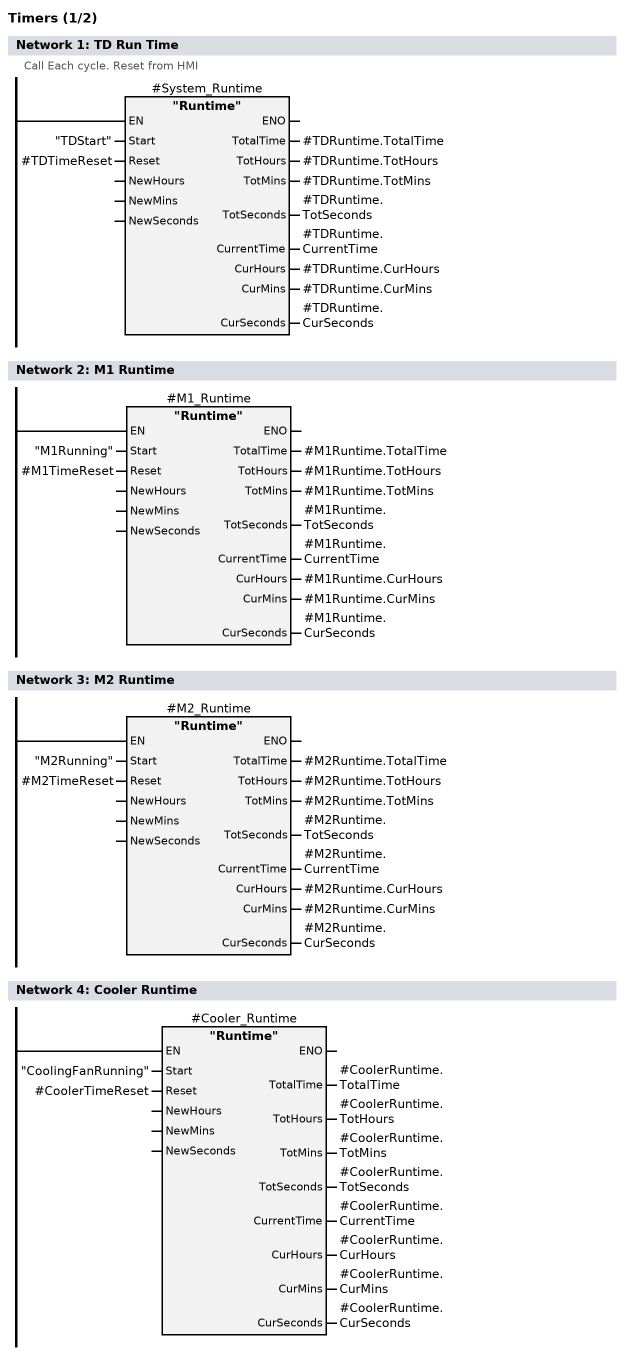
   RUNG wire#powerrail
      #System_Runtime(Start := "TDStart", Reset := #TDTimeReset, NewHours :=, NewMins :=, NewSeconds :=, TotalTime => #TDRuntime.TotalTime, TotHours => #TDRuntime.TotHours, TotMins => #TDRuntime.TotMins, TotSeconds => #TDRuntime.TotSeconds, CurrentTime => #TDRuntime.CurrentTime, CurHours => #TDRuntime.CurHours, CurMins => #TDRuntime.CurMins, CurSeconds => #TDRuntime.CurSeconds)
   END_RUNG
   // the same network as SCL:
   #System_Runtime(Start := "TDStart",   // "Runtime"
                   Reset := #TDTimeReset,
                   TotalTime => #TDRuntime.TotalTime,
                   TotHours => #TDRuntime.TotHours,
                   TotMins => #TDRuntime.TotMins,
                   TotSeconds => #TDRuntime.TotSeconds,
                   CurrentTime => #TDRuntime.CurrentTime,
                   CurHours => #TDRuntime.CurHours,
                   CurMins => #TDRuntime.CurMins,
                   CurSeconds => #TDRuntime.CurSeconds);
END_REGION

REGION Network 2: M1 Runtime
   RUNG wire#powerrail
      #M1_Runtime(Start := "M1Running", Reset := #M1TimeReset, NewHours :=, NewMins :=, NewSeconds :=, TotalTime => #M1Runtime.TotalTime, TotHours => #M1Runtime.TotHours, TotMins => #M1Runtime.TotMins, TotSeconds => #M1Runtime.TotSeconds, CurrentTime => #M1Runtime.CurrentTime, CurHours => #M1Runtime.CurHours, CurMins => #M1Runtime.CurMins, CurSeconds => #M1Runtime.CurSeconds)
   END_RUNG
   // the same network as SCL:
   #M1_Runtime(Start := "M1Running",   // "Runtime"
               Reset := #M1TimeReset,
               TotalTime => #M1Runtime.TotalTime,
               TotHours => #M1Runtime.TotHours,
               TotMins => #M1Runtime.TotMins,
               TotSeconds => #M1Runtime.TotSeconds,
               CurrentTime => #M1Runtime.CurrentTime,
               CurHours => #M1Runtime.CurHours,
               CurMins => #M1Runtime.CurMins,
               CurSeconds => #M1Runtime.CurSeconds);
END_REGION

REGION Network 3: M2 Runtime
   RUNG wire#powerrail
      #M2_Runtime(Start := "M2Running", Reset := #M2TimeReset, NewHours :=, NewMins :=, NewSeconds :=, TotalTime => #M2Runtime.TotalTime, TotHours => #M2Runtime.TotHours, TotMins => #M2Runtime.TotMins, TotSeconds => #M2Runtime.TotSeconds, CurrentTime => #M2Runtime.CurrentTime, CurHours => #M2Runtime.CurHours, CurMins => #M2Runtime.CurMins, CurSeconds => #M2Runtime.CurSeconds)
   END_RUNG
   // the same network as SCL:
   #M2_Runtime(Start := "M2Running",   // "Runtime"
               Reset := #M2TimeReset,
               TotalTime => #M2Runtime.TotalTime,
               TotHours => #M2Runtime.TotHours,
               TotMins => #M2Runtime.TotMins,
               TotSeconds => #M2Runtime.TotSeconds,
               CurrentTime => #M2Runtime.CurrentTime,
               CurHours => #M2Runtime.CurHours,
               CurMins => #M2Runtime.CurMins,
               CurSeconds => #M2Runtime.CurSeconds);
END_REGION

REGION Network 4: Cooler Runtime
   RUNG wire#powerrail
      #Cooler_Runtime(Start := "CoolingFanRunning", Reset := #CoolerTimeReset, NewHours :=, NewMins :=, NewSeconds :=, TotalTime => #CoolerRuntime.TotalTime, TotHours => #CoolerRuntime.TotHours, TotMins => #CoolerRuntime.TotMins, TotSeconds => #CoolerRuntime.TotSeconds, CurrentTime => #CoolerRuntime.CurrentTime, CurHours => #CoolerRuntime.CurHours, CurMins => #CoolerRuntime.CurMins, CurSeconds => #CoolerRuntime.CurSeconds)
   END_RUNG
   // the same network as SCL:
   #Cooler_Runtime(Start := "CoolingFanRunning",   // "Runtime"
                   Reset := #CoolerTimeReset,
                   TotalTime => #CoolerRuntime.TotalTime,
                   TotHours => #CoolerRuntime.TotHours,
                   TotMins => #CoolerRuntime.TotMins,
                   TotSeconds => #CoolerRuntime.TotSeconds,
                   CurrentTime => #CoolerRuntime.CurrentTime,
                   CurHours => #CoolerRuntime.CurHours,
                   CurMins => #CoolerRuntime.CurMins,
                   CurSeconds => #CoolerRuntime.CurSeconds);
END_REGION

REGION Network 5: Aux Pump Runtime
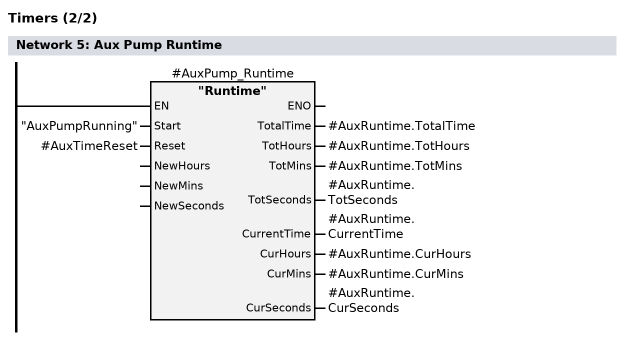
   RUNG wire#powerrail
      #AuxPump_Runtime(Start := "AuxPumpRunning", Reset := #AuxTimeReset, NewHours :=, NewMins :=, NewSeconds :=, TotalTime => #AuxRuntime.TotalTime, TotHours => #AuxRuntime.TotHours, TotMins => #AuxRuntime.TotMins, TotSeconds => #AuxRuntime.TotSeconds, CurrentTime => #AuxRuntime.CurrentTime, CurHours => #AuxRuntime.CurHours, CurMins => #AuxRuntime.CurMins, CurSeconds => #AuxRuntime.CurSeconds)
   END_RUNG
   // the same network as SCL:
   #AuxPump_Runtime(Start := "AuxPumpRunning",   // "Runtime"
                    Reset := #AuxTimeReset,
                    TotalTime => #AuxRuntime.TotalTime,
                    TotHours => #AuxRuntime.TotHours,
                    TotMins => #AuxRuntime.TotMins,
                    TotSeconds => #AuxRuntime.TotSeconds,
                    CurrentTime => #AuxRuntime.CurrentTime,
                    CurHours => #AuxRuntime.CurHours,
                    CurMins => #AuxRuntime.CurMins,
                    CurSeconds => #AuxRuntime.CurSeconds);
END_REGION
END_FUNCTION_BLOCK

FUNCTION_BLOCK "Runtime"   // FB124, LAD
{ S7_Optimized_Access := 'TRUE' }
// Written By Kristopher Gimenez March 3rd,2023
// 
// This block and its DB will perform a runtime counter and outputs total runtime in Hours, Minutes and Seconds
// stored: AutoNumber false, MemoryReserve 100, SetENOAutomatically false
   VAR_INPUT
      Start : Bool;
      Reset : Bool;
      NewHours : DInt;
      NewMins : DInt;
      NewSeconds : DInt;
   END_VAR
   VAR_OUTPUT
      TotalTime : DInt;
      TotHours : DInt;
      TotMins : DInt;
      TotSeconds : DInt;
      CurrentTime : DInt;   // Current Time in Seconds
      CurHours : DInt;
      CurMins : DInt;
      CurSeconds : DInt;
   END_VAR
   VAR
      StartTrig : Bool;
      StartTime : DInt;
      Runtime_TONR { S7_SetPoint := 'True'} : TONR_TIME;
      TimerReset { ExternalAccessible := 'False'; ExternalVisible := 'False'; ExternalWritable := 'False'} : Bool;
      CurrentIECTime : Time;
      NewTime : DInt;   // New Time in seconds to reset to base on inputs
   END_VAR
   VAR_TEMP
      TempDInt : DInt;
      NewHoursInSec : DInt;
      NewMinsInSec : DInt;
   END_VAR
   VAR_TEMP   // added for the SCL form of the ladder/FBD networks
      _w1 : Bool;
   END_VAR
BEGIN

REGION Network 1: Start
   // When Starting store Total as Start Value
   // Reset Current Runtime
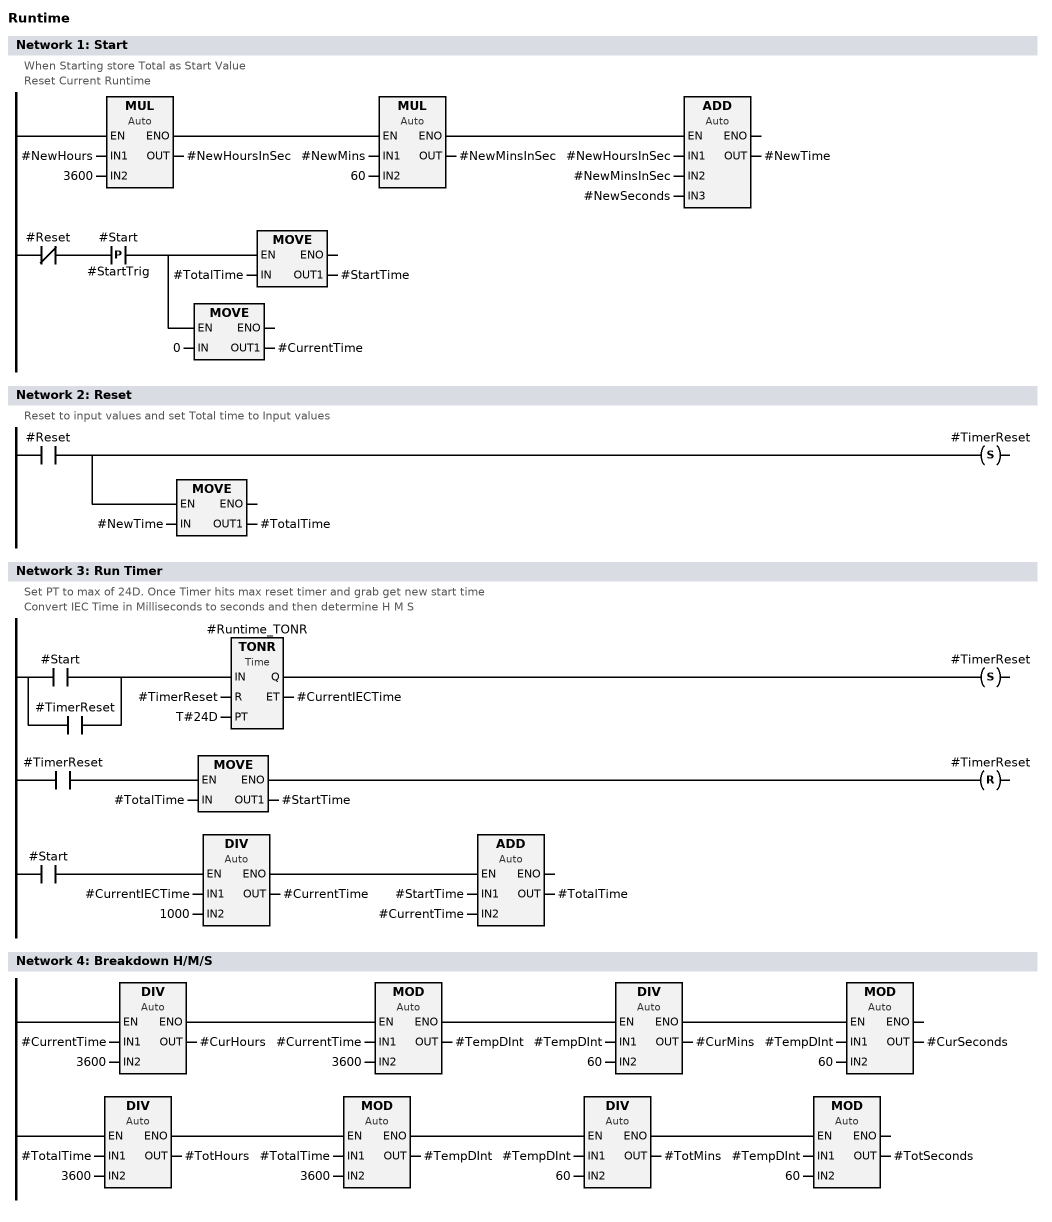
   RUNG wire#powerrail
      Mul(in1 := #NewHours, in2 := 3600, out => #NewHoursInSec)
      Mul(in1 := #NewMins, in2 := 60, out => #NewMinsInSec)
      Add(in1 := #NewHoursInSec, in2 := #NewMinsInSec, in3 := #NewSeconds, out => #NewTime)
   END_RUNG
   RUNG wire#powerrail
      I_Contact( #Reset )
      P_Contact(operand := #Start, bit := #StartTrig)
      wire#w1
      Move(in := #TotalTime, out1 => #StartTime)
   END_RUNG
   RUNG wire#w1
      Move(in := 0, out1 => #CurrentTime)
   END_RUNG
   // the same network as SCL:
   #NewHoursInSec := #NewHours * 3600;
   #NewMinsInSec := #NewMins * 60;
   #NewTime := #NewHoursInSec + #NewMinsInSec + #NewSeconds;
   #_w1 := NOT #Reset AND #Start AND NOT #StartTrig;   // rising edge of #Start
   #StartTrig := #Start;
   IF #_w1 THEN
       #StartTime := #TotalTime;
       #CurrentTime := 0;
   END_IF;
END_REGION

REGION Network 2: Reset
   // Reset to input values and set Total time to Input values
   RUNG wire#powerrail
      Contact( #Reset )
      wire#w1
      S_Coil( #TimerReset )
   END_RUNG
   RUNG wire#w1
      Move(in := #NewTime, out1 => #TotalTime)
   END_RUNG
   // the same network as SCL:
   IF #Reset THEN
       #TimerReset := TRUE;
       #TotalTime := #NewTime;
   END_IF;
END_REGION

REGION Network 3: Run Timer
   // Set PT to max of 24D. Once Timer hits max reset timer and grab get new start time
   // Convert IEC Time in Milliseconds to seconds and then determine H M S
   RUNG wire#powerrail
      Contact( #Start )
      wire#w1
      { S7_Templates := "time_type := Time" } #Runtime_TONR.TONR(r := #TimerReset, pt := T#24D, et => #CurrentIECTime)
      S_Coil( #TimerReset )
   END_RUNG
   RUNG wire#powerrail
      Contact( #TimerReset )
   END_RUNG wire#w1
   RUNG wire#powerrail
      Contact( #TimerReset )
      Move(in := #TotalTime, out1 => #StartTime)
      R_Coil( #TimerReset )
   END_RUNG
   RUNG wire#powerrail
      Contact( #Start )
      Div(in1 := #CurrentIECTime, in2 := 1000, out => #CurrentTime)
      Add(in1 := #StartTime, in2 := #CurrentTime, out => #TotalTime)
   END_RUNG
   // the same network as SCL:
   #Runtime_TONR(IN := #Start OR #TimerReset, R := #TimerReset, PT := T#24D, ET => #CurrentIECTime);   // TONR
   IF #Runtime_TONR.Q THEN #TimerReset := TRUE; END_IF;
   IF #TimerReset THEN
       #StartTime := #TotalTime;
       #TimerReset := FALSE;
   END_IF;
   IF #Start THEN
       #CurrentTime := #CurrentIECTime / 1000;
       #TotalTime := #StartTime + #CurrentTime;
   END_IF;
END_REGION

REGION Network 4: Breakdown H/M/S
   RUNG wire#powerrail
      Div(in1 := #CurrentTime, in2 := 3600, out => #CurHours)
      Mod(in1 := #CurrentTime, in2 := 3600, out => #TempDInt)
      Div(in1 := #TempDInt, in2 := 60, out => #CurMins)
      Mod(in1 := #TempDInt, in2 := 60, out => #CurSeconds)
   END_RUNG
   RUNG wire#powerrail
      Div(in1 := #TotalTime, in2 := 3600, out => #TotHours)
      Mod(in1 := #TotalTime, in2 := 3600, out => #TempDInt)
      Div(in1 := #TempDInt, in2 := 60, out => #TotMins)
      Mod(in1 := #TempDInt, in2 := 60, out => #TotSeconds)
   END_RUNG
   // the same network as SCL:
   #CurHours := #CurrentTime / 3600;
   #TempDInt := #CurrentTime MOD 3600;
   #CurMins := #TempDInt / 60;
   #CurSeconds := #TempDInt MOD 60;
   #TotHours := #TotalTime / 3600;
   #TempDInt := #TotalTime MOD 3600;
   #TotMins := #TempDInt / 60;
   #TotSeconds := #TempDInt MOD 60;
END_REGION
END_FUNCTION_BLOCK

FUNCTION "MapConsoleOutputs" : Void
{ S7_Optimized_Access := 'TRUE' }
VERSION : 0.1

BEGIN
	(* #MapConsoleOutputs Written BY Kristopher Gimenez January 23,2023
	This block is will map the output variables and convert raw signals into measured values
	*)
	
	
	
	//Slot 4 16x Digital Outputs
	"Console_Out".Slot4.Ch0 :="PTOLED";
	"Console_Out".Slot4.Ch1 := "HPUFaultLED";
	"Console_Out".Slot4.Ch2 := "TDFlushFaultLED";
	"Console_Out".Slot4.Ch3 := "BUWClLED";
	"Console_Out".Slot4.Ch4 := "TDEnLED";
	"Console_Out".Slot4.Ch5 := "ConLowPurgeLED";
	"Console_Out".Slot4.Ch6 := "MSVClLED";
	"Console_Out".Slot4.Ch7 := "QuillLockLED";
	"Console_Out".Slot4.Ch8 := "ElevClLED";
	"Console_Out".Slot4.Ch9 := "Horn";
	"Console_Out".Slot4.Ch10 := "MSVClInt";
	"Console_Out".Slot4.Ch11 := "BUWClInt";
	(*Spare Outputs
	"Console_Out".Slot4.Ch12 := ;
	"Console_Out".Slot4.Ch13 := ;
	"Console_Out".Slot4.Ch14 := ;
	"Console_Out".Slot4.Ch15 := ;
	*)
	
	
	
	
	//Slot 5 4 x AQ U/I
	"AoUI_Scaling"(Measured:="DrillRecTorqFtLbs",
	               Max:=40000.0,
	               Min:=0,
	               s7Raw=>"DrillRecTorqRaw",
	               mAOutput=>"DrillRecTorqmA"); //4-20ma = 0-40 000 ft-lbs
	"AoUI_Scaling"(Measured:="DrillRecRPM",
	               Max:=200.0,
	               Min:=0,
	               s7Raw=>"DrillRecRPMRaw",
	               mAOutput=>"DrillRecRPMmA");// 4-20ma = 0-200 RPM
	
	
	"Console_Out".Slot5.Ch0 := "DrillRecTorqRaw";
	"Console_Out".Slot5.Ch1 := ("DrillRecRPMRaw");
END_FUNCTION

FUNCTION "AoUI_Scaling" : Void
{ S7_Optimized_Access := 'TRUE' }
VERSION : 0.1
   VAR_INPUT 
      Measured : Real;   // Measured
      Max : Real;   // Maximum mreasured value of output
      Min : Real;   // Minimum measured value of output
   END_VAR

   VAR_OUTPUT 
      s7Raw : Int;   // Raw Outputs to card 
      mAOutput : Real;   // 4-20ma Output based on raw outputs
   END_VAR


BEGIN
	(* #AoUI_Scaling Written BY Kristopher Gimenez January 23,2023
	This block is used to convert a Measured value into a PS7 analog output and the corresponding 4-20mA signal based on Scale and Offset. 
	*)
	
	
	#s7Raw := REAL_TO_INT((#Measured-#Min)/(#Max - #Min) * 27648);
	#mAOutput := ((#Measured-#Min)/(#Max-#Min) * 16.0) + 4.0;
	
	
END_FUNCTION

FUNCTION "MapHPUOutputs" : Void
{ S7_Optimized_Access := 'TRUE' }
VERSION : 0.1

BEGIN
	(* #MapHPUOutputs Written BY Kristopher Gimenez January 19,2023
	This block is will map the input variables and convert raw signals into measured values
	*)
	//HPU Slot2 TM Count Encoder Outputs
	"HPU_Out".Slot2.SW_GATE := "SwitchSWGATE"; //Enable the counter
	"HPU_Out".Slot2.SET_DIR:= "RotaryEncInvDir";
	"HPU_Out".Slot2.SLOT_0 := "RotEncSlot0";
	"HPU_Out".Slot2.SLOT_1 := "RotEncSlot1";
	"HPU_Out".Slot2.LD_SLOT_0_1 := "RotEncLDSlot";//assign loading bytes
	"HPU_Out".Slot2.RES_EVENT := "RotEncPosReset";//reset event flags if position is being res
	
	
	//Slot 7 TM Pulse
	//Channel 0 TD P1 Fwd
	"TDFwdPress1Raw" := "AoP_mA2Raw_2A"("TDFwdPress1mA");
	"HPU_Out".Slot7.Ch0.OUTPUT_VALUE := "TDFwdPress1Raw";//assign output value
	"HPU_Out".Slot7.Ch0.SW_ENABLE :="TDFwdPress1En"; //used to enabled output
	"HPU_Out".Slot7.Ch0.DITHER := "TDFwdPress1En"; //enable Dither - Currently enabling with the output. 
	"HPU_Out".Slot7.Ch0.TM_CTRL_DQ :=1;//enable technology control of outputs 
	//Channel 1 TD P1 Rev
	"TDRevPress1Raw" := "AoP_mA2Raw_2A"("TDRevPress1mA");
	"HPU_Out".Slot7.Ch1.OUTPUT_VALUE := "TDRevPress1Raw";//assign output value
	"HPU_Out".Slot7.Ch1.SW_ENABLE := "TDRevPress1En"; //used to enabled output
	"HPU_Out".Slot7.Ch1.DITHER := "TDRevPress1En"; //enable Dither - Currently enabling with the output. 
	"HPU_Out".Slot7.Ch1.TM_CTRL_DQ := 1;//enable technology control of outputs 
	
	
	
	//Slot 8 TM Pulse
	//Channel 0 TD P2 FWD
	"TDFwdPress2Raw" := "AoP_mA2Raw_2A"("TDFwdPress2mA");
	"HPU_Out".Slot8.Ch0.OUTPUT_VALUE := "TDFwdPress2Raw";//assign output value
	"HPU_Out".Slot8.Ch0.SW_ENABLE := "TDFwdPress2En"; //used to enabled output
	"HPU_Out".Slot8.Ch0.DITHER := "TDFwdPress2En"; //enable Dither - Currently enabling with the output. 
	"HPU_Out".Slot8.Ch0.TM_CTRL_DQ := 1;//enable technology control of outputs 
	
	//Channel 1 TD P2 Rev
	"TDRevPress2Raw" := "AoP_mA2Raw_2A"("TDRevPress2mA");
	"HPU_Out".Slot8.Ch1.OUTPUT_VALUE := "TDRevPress2Raw";//assign output value
	"HPU_Out".Slot8.Ch1.SW_ENABLE := "TDRevPress2En"; //used to enabled output
	"HPU_Out".Slot8.Ch1.DITHER := "TDRevPress2En"; //enable Dither - Currently enabling with the output. 
	"HPU_Out".Slot8.Ch1.TM_CTRL_DQ := 1;//enable technology control of outputs 
	
	
	//Slot 9 TM Pulse
	//Channel 0 TD Torq
	"TDTorqPressRaw" := "AoP_mA2Raw_2A"("TDTorqPressmA");
	"HPU_Out".Slot9.Ch0.OUTPUT_VALUE := "TDTorqPressRaw";//assign output value
	"HPU_Out".Slot9.Ch0.SW_ENABLE := "TDTorqPressEn"; //used to enabled output
	"HPU_Out".Slot9.Ch0.DITHER := "TDTorqPressEn"; //enable Dither - Currently enabling with the output. 
	"HPU_Out".Slot9.Ch0.TM_CTRL_DQ := 1;//enable technology control of outputs 
	//Slot 9 TM Pulse
	//Channel 1 TD P1 Rev
	//"TDRevPress1Raw" := "AoP_mA2Raw_2A"("TDRevPress1mA");
	//"HPU_Out".Slot9.Ch1.OUTPUT_VALUE := "TDRevPress1Raw";//assign output value
	//"HPU_Out".Slot9.Ch1.SW_ENABLE := "TDRevPress1En"; //used to enabled output
	//"HPU_Out".Slot9.Ch1.DITHER := "TDRevPress1En"; //enable Dither - Currently enabling with the output. 
	//"HPU_Out".Slot9.Ch1.TM_CTRL_DQ := 1;//enable technology control of outputs 
	
	//Slot 10 DO Relay x 4
	"HPU_Out".Slot10.Ch0 := "M1Start";
	"HPU_Out".Slot10.Ch1 := "M2Start";
	"HPU_Out".Slot10.Ch2 := "CoolingFanStart";
	"HPU_Out".Slot10.Ch3 := "AuxPumpStart";
	
	//Slot 11 DO Relay x 4
	"HPU_Out".Slot11.Ch0 := "LinkExtSol";
	"HPU_Out".Slot11.Ch1 := "LinkRetSol";
	"HPU_Out".Slot11.Ch2 := "LinkFloatSol";
	//"HPU_Out".Slot11.Ch3 := ;Spare
	
	
	//Slot 12 DO Relay x 4
	"HPU_Out".Slot12.Ch0 := "BUWClSol";
	"HPU_Out".Slot12.Ch1 := "BUWDnSol";
	"HPU_Out".Slot12.Ch2 := "BUWUpSol";
	"HPU_Out".Slot12.Ch3 := "BUWOpSol";
	
	
	//Slot 13 DO Relay x 4
	"HPU_Out".Slot13.Ch0 := "LSHT_Sol";
	"HPU_Out".Slot13.Ch1 := "HSLT_Sol";
	"HPU_Out".Slot13.Ch2 := "ElevClSol";
	"HPU_Out".Slot13.Ch3 := "ElevOpSol";
	
	
	//Slot 14 DO Relay x 4
	"HPU_Out".Slot14.Ch0 := "HandlerFWDSol";
	"HPU_Out".Slot14.Ch1 := "HandlerREVSol";
	"HPU_Out".Slot14.Ch2 := "MSVOpSol";
	"HPU_Out".Slot14.Ch3 := "MSVClSol";
	
	
	//Slot 15 DO Relay x 4
	"HPU_Out".Slot15.Ch0 := "HourMeterOn";
	"HPU_Out".Slot15.Ch1 := "FailSafeEnSol";
	"HPU_Out".Slot15.Ch2 := "AuxUnloaderSol";
	"HPU_Out".Slot15.Ch3 := "BypassValveSol";
	
	
	//Slot 16 DO Relay x 4
	"HPU_Out".Slot16.Ch0 := "TDExtSol";
	"HPU_Out".Slot16.Ch1 := "TDRetSol";
	"HPU_Out".Slot16.Ch2 := "HotOilControlSol";
	"HPU_Out".Slot16.Ch3 := "BOControlSol";
	
	//Slot 17 DO Relay x 4
	(*Spare Outputs
	"HPU_Out".Slot17.Ch0 := ;
	"HPU_Out".Slot17.Ch1 := ;
	"HPU_Out".Slot18.Ch2 := ;
	"HPU_Out".Slot18.Ch3 := ;
	*)
END_FUNCTION

FUNCTION "AoP_mA2Raw_2A" : UDInt
{ S7_Optimized_Access := 'TRUE' }
VERSION : 0.1
   VAR_INPUT 
      Realnput : Real;
   END_VAR


BEGIN
	(* #AoP_ma2Raw_2A Written BY Kristopher Gimenez January 23,2023
	This block is used to convert a mA signal  output signal to a Raw. Note 0-2A = 27648 pulse output.
	*)
	
	
	#AoP_mA2Raw_2A := REAL_TO_UDINT(#Realnput/2000* 27648.0);
	
	
END_FUNCTION

ORGANIZATION_BLOCK "Startup"   // OB100, LAD, Startup
TITLE = "Complete Restart"
{ S7_Optimized_Access := 'TRUE' }
// stored: SetENOAutomatically false
   VAR_INPUT
      LostRetentive : Bool;   // True if retentive data are lost
      LostRTC : Bool;   // True if date and time are lost
   END_VAR
   VAR_TEMP
      RetVal : Int;
      BusyStatus : Bool;
   END_VAR
   VAR_TEMP   // added for the SCL form of the ladder/FBD networks
      _w1 : Bool;
   END_VAR
BEGIN

REGION Network 1: Verify Settings
   // Check settings on startup
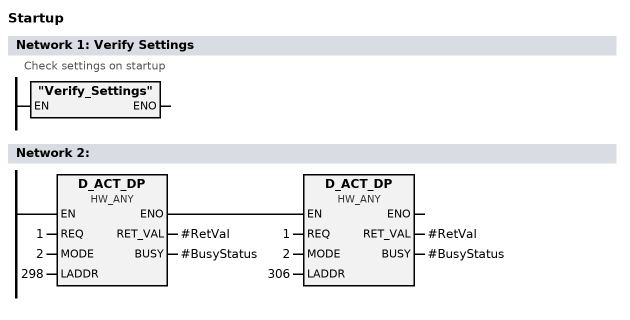
   RUNG wire#powerrail
      "Verify_Settings"()
   END_RUNG
   // the same network as SCL:
   "Verify_Settings"();
END_REGION

REGION Network 2
   RUNG wire#powerrail
      { S7_Templates := "[laddr_type := HW_ANY, mode_type := USInt]" } D_ACT_DP(REQ := 1, MODE := 2, LADDR := 298, RET_VAL => #RetVal, BUSY => #BusyStatus)
      { S7_Templates := "[laddr_type := HW_ANY, mode_type := USInt]" } D_ACT_DP(REQ := 1, MODE := 2, LADDR := 306, RET_VAL => #RetVal, BUSY => #BusyStatus)
   END_RUNG
   // the same network as SCL:
   #RetVal := D_ACT_DP(REQ := 1, MODE := 2, LADDR := 298, BUSY => #BusyStatus, ENO => #_w1);
   IF #_w1 THEN #RetVal := D_ACT_DP(REQ := 1, MODE := 2, LADDR := 306, BUSY => #BusyStatus); END_IF;
END_REGION
END_ORGANIZATION_BLOCK

FUNCTION "Verify_Settings" : Void   // FC21, LAD
{ S7_Optimized_Access := 'TRUE' }
// Written BY Kristopher Gimenez February 9th, 2023
// This block is used to check the settings are within limits and adjust as needed
// stored: AutoNumber false, SetENOAutomatically false
BEGIN

REGION Network 1: Alpha Values
   // All alpha filter values between 0-1
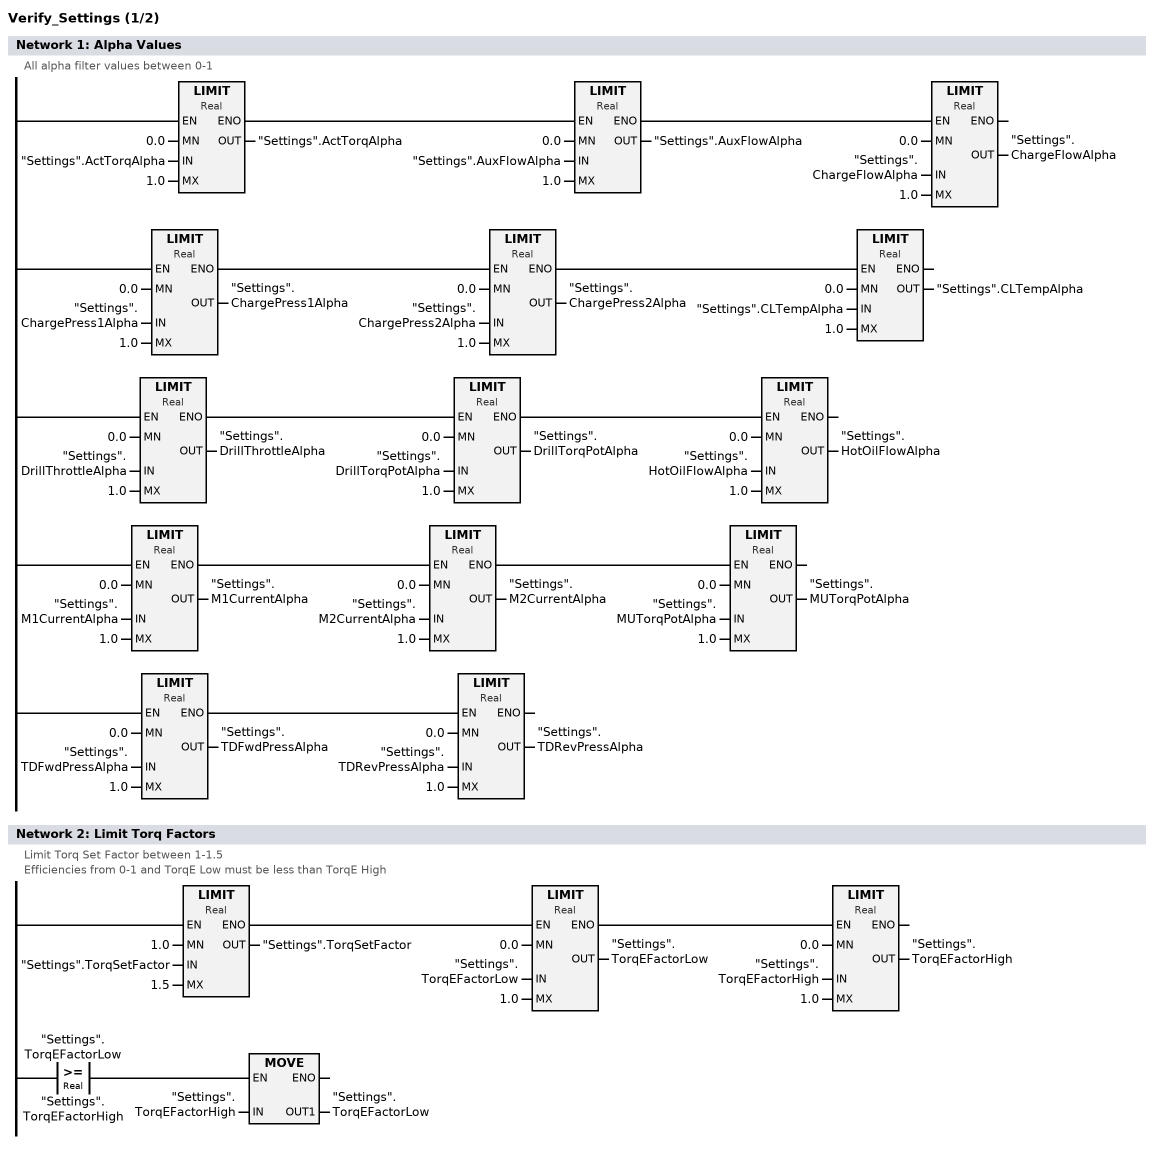
   RUNG wire#powerrail
      { S7_Templates := "value_type := Real" } Limit(mn := 0.0, in := "Settings".ActTorqAlpha, mx := 1.0, out => "Settings".ActTorqAlpha)
      { S7_Templates := "value_type := Real" } Limit(mn := 0.0, in := "Settings".AuxFlowAlpha, mx := 1.0, out => "Settings".AuxFlowAlpha)
      { S7_Templates := "value_type := Real" } Limit(mn := 0.0, in := "Settings".ChargeFlowAlpha, mx := 1.0, out => "Settings".ChargeFlowAlpha)
   END_RUNG
   RUNG wire#powerrail
      { S7_Templates := "value_type := Real" } Limit(mn := 0.0, in := "Settings".ChargePress1Alpha, mx := 1.0, out => "Settings".ChargePress1Alpha)
      { S7_Templates := "value_type := Real" } Limit(mn := 0.0, in := "Settings".ChargePress2Alpha, mx := 1.0, out => "Settings".ChargePress2Alpha)
      { S7_Templates := "value_type := Real" } Limit(mn := 0.0, in := "Settings".CLTempAlpha, mx := 1.0, out => "Settings".CLTempAlpha)
   END_RUNG
   RUNG wire#powerrail
      { S7_Templates := "value_type := Real" } Limit(mn := 0.0, in := "Settings".DrillThrottleAlpha, mx := 1.0, out => "Settings".DrillThrottleAlpha)
      { S7_Templates := "value_type := Real" } Limit(mn := 0.0, in := "Settings".DrillTorqPotAlpha, mx := 1.0, out => "Settings".DrillTorqPotAlpha)
      { S7_Templates := "value_type := Real" } Limit(mn := 0.0, in := "Settings".HotOilFlowAlpha, mx := 1.0, out => "Settings".HotOilFlowAlpha)
   END_RUNG
   RUNG wire#powerrail
      { S7_Templates := "value_type := Real" } Limit(mn := 0.0, in := "Settings".M1CurrentAlpha, mx := 1.0, out => "Settings".M1CurrentAlpha)
      { S7_Templates := "value_type := Real" } Limit(mn := 0.0, in := "Settings".M2CurrentAlpha, mx := 1.0, out => "Settings".M2CurrentAlpha)
      { S7_Templates := "value_type := Real" } Limit(mn := 0.0, in := "Settings".MUTorqPotAlpha, mx := 1.0, out => "Settings".MUTorqPotAlpha)
   END_RUNG
   RUNG wire#powerrail
      { S7_Templates := "value_type := Real" } Limit(mn := 0.0, in := "Settings".TDFwdPressAlpha, mx := 1.0, out => "Settings".TDFwdPressAlpha)
      { S7_Templates := "value_type := Real" } Limit(mn := 0.0, in := "Settings".TDRevPressAlpha, mx := 1.0, out => "Settings".TDRevPressAlpha)
   END_RUNG
   // the same network as SCL:
   "Settings".ActTorqAlpha := LIMIT(MN := 0.0, IN := "Settings".ActTorqAlpha, MX := 1.0);
   "Settings".AuxFlowAlpha := LIMIT(MN := 0.0, IN := "Settings".AuxFlowAlpha, MX := 1.0);
   "Settings".ChargeFlowAlpha := LIMIT(MN := 0.0, IN := "Settings".ChargeFlowAlpha, MX := 1.0);
   "Settings".ChargePress1Alpha := LIMIT(MN := 0.0, IN := "Settings".ChargePress1Alpha, MX := 1.0);
   "Settings".ChargePress2Alpha := LIMIT(MN := 0.0, IN := "Settings".ChargePress2Alpha, MX := 1.0);
   "Settings".CLTempAlpha := LIMIT(MN := 0.0, IN := "Settings".CLTempAlpha, MX := 1.0);
   "Settings".DrillThrottleAlpha := LIMIT(MN := 0.0, IN := "Settings".DrillThrottleAlpha, MX := 1.0);
   "Settings".DrillTorqPotAlpha := LIMIT(MN := 0.0, IN := "Settings".DrillTorqPotAlpha, MX := 1.0);
   "Settings".HotOilFlowAlpha := LIMIT(MN := 0.0, IN := "Settings".HotOilFlowAlpha, MX := 1.0);
   "Settings".M1CurrentAlpha := LIMIT(MN := 0.0, IN := "Settings".M1CurrentAlpha, MX := 1.0);
   "Settings".M2CurrentAlpha := LIMIT(MN := 0.0, IN := "Settings".M2CurrentAlpha, MX := 1.0);
   "Settings".MUTorqPotAlpha := LIMIT(MN := 0.0, IN := "Settings".MUTorqPotAlpha, MX := 1.0);
   "Settings".TDFwdPressAlpha := LIMIT(MN := 0.0, IN := "Settings".TDFwdPressAlpha, MX := 1.0);
   "Settings".TDRevPressAlpha := LIMIT(MN := 0.0, IN := "Settings".TDRevPressAlpha, MX := 1.0);
END_REGION

REGION Network 2: Limit Torq Factors
   // Limit Torq Set Factor between 1-1.5
   // Efficiencies from 0-1 and TorqE Low must be less than TorqE High
   RUNG wire#powerrail
      { S7_Templates := "value_type := Real" } Limit(mn := 1.0, in := "Settings".TorqSetFactor, mx := 1.5, out => "Settings".TorqSetFactor)
      { S7_Templates := "value_type := Real" } Limit(mn := 0.0, in := "Settings".TorqEFactorLow, mx := 1.0, out => "Settings".TorqEFactorLow)
      { S7_Templates := "value_type := Real" } Limit(mn := 0.0, in := "Settings".TorqEFactorHigh, mx := 1.0, out => "Settings".TorqEFactorHigh)
   END_RUNG
   RUNG wire#powerrail
      { S7_Templates := "SrcType := Real" } GE_Contact(in1 := "Settings".TorqEFactorLow, in2 := "Settings".TorqEFactorHigh)
      Move(in := "Settings".TorqEFactorHigh, out1 => "Settings".TorqEFactorLow)
   END_RUNG
   // the same network as SCL:
   "Settings".TorqSetFactor := LIMIT(MN := 1.0, IN := "Settings".TorqSetFactor, MX := 1.5);
   "Settings".TorqEFactorLow := LIMIT(MN := 0.0, IN := "Settings".TorqEFactorLow, MX := 1.0);
   "Settings".TorqEFactorHigh := LIMIT(MN := 0.0, IN := "Settings".TorqEFactorHigh, MX := 1.0);
   IF "Settings".TorqEFactorLow >= "Settings".TorqEFactorHigh THEN
       "Settings".TorqEFactorLow := "Settings".TorqEFactorHigh;
   END_IF;
END_REGION

REGION Network 3: Verify BO Setting
   // BO Spin Factor from 1-2
   // Shift RPM from 1 to Speed limit
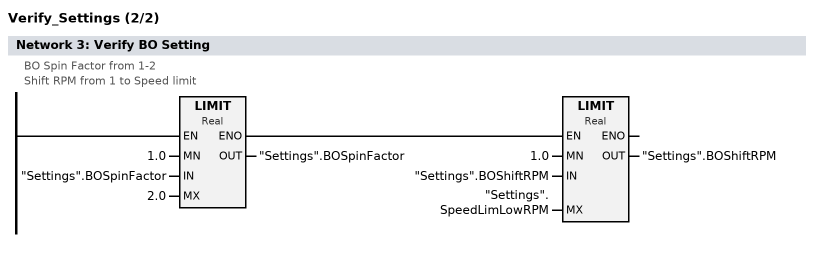
   RUNG wire#powerrail
      { S7_Templates := "value_type := Real" } Limit(mn := 1.0, in := "Settings".BOSpinFactor, mx := 2.0, out => "Settings".BOSpinFactor)
      { S7_Templates := "value_type := Real" } Limit(mn := 1.0, in := "Settings".BOShiftRPM, mx := "Settings".SpeedLimLowRPM, out => "Settings".BOShiftRPM)
   END_RUNG
   // the same network as SCL:
   "Settings".BOSpinFactor := LIMIT(MN := 1.0, IN := "Settings".BOSpinFactor, MX := 2.0);
   "Settings".BOShiftRPM := LIMIT(MN := 1.0, IN := "Settings".BOShiftRPM, MX := "Settings".SpeedLimLowRPM);
END_REGION
END_FUNCTION

FUNCTION_BLOCK "Block_1"
{ S7_Optimized_Access := 'TRUE' }
VERSION : 0.1
   VAR_INPUT 
      Input_1 : Bool;
   END_VAR

   VAR 
      Test_Mode : Word;
      "Counter" : Word := 0;
      Delay_Timer {InstructionName := 'TON_TIME'; LibVersion := '1.0'} : TON_TIME;
      TurnOnOffTimer { S7_SetPoint := 'True'} : Bool;
   END_VAR

   VAR_TEMP 
      PTOLED : Bool;
      HpuFaultLed : Bool;
      BUWCLLED : Bool;
      QuillLockLED : Bool;
      TDEnableLed : Bool;
      MSVClLED : Bool;
      ElevatorCLLED : Bool;
   END_VAR

   VAR CONSTANT 
      AuxByPassMode : Word := 2;
      AuxByPassModeDone : Word := 3;
      TDEnableMode : Word := 4;
      TDEnableModeDone : Word := 5;
      BUWAutoClHoldingMode : Word := 6;
      BUWAutoClHoldingModeDone : Word := 7;
      QuillLockMode : Word := 8;
      QuillLockModeDone : Word := 9;
      MudSaverOpenMode : Word := 10;
      MudSaverCloseMode : Word := 11;
      MudSaverAutoMode : Word := 12;
      MudSaveModeDone : Word := 13;
      ElevCloseMode : Word := 14;
      ElevOpenMode : Word := 15;
      "MudSaverPumpRuningMode-0" : Word := 16;
      "MudSaverPumpRuningMode-1" : Word := 17;
   END_VAR


BEGIN
	//#Test_Mode := #AuxByPassMode;
	//#Test_Mode := #AuxByPassModeDone;
	//#Test_Mode := #TDEnableMode;
	//#Test_Mode := #BUWAutoClHoldingModeDone;
	//#Test_Mode := #QuillLockMode;
	//#Test_Mode := #QuillLockModeDone;
	//#Test_Mode := #MudSaverCloseMode;
	//#Test_Mode := #MudSaverOpenMode;
	//#Test_Mode := #MudSaverAutoMode;
	//#Test_Mode := #"MudSaverPumpRuningMode-0";  //close
	//#Test_Mode := #"MudSaverPumpRuningMode-1"; //open
	#Test_Mode := #ElevOpenMode;
	//#Test_Mode := #ElevCloseMode;
	IF #Test_Mode = #AuxByPassMode THEN  //AuxByPass Mode
	    "Console_In".Slot1.Ch1 := 1; //TDAuxSw
	    "Console_In".Slot1.Ch3 := 0; //TDEnableSw 
	    "HPU_In".Slot3.Ch0 := 1; //AuxPumpRunning feedback
	    "Console_In".Slot1.Ch8 := 1; //Quill lock,    //Control bit
	    "Console_In".Slot2.Ch4 := 1;//PTO_sw, After PTO, BUW Closed //Control bit
	END_IF;
	IF #Test_Mode = #AuxByPassModeDone THEN
	        
	        "Console_In".Slot1.Ch8 := 0; //Quill lock,    //Control bit
	        "Console_In".Slot2.Ch4 := 0;//PTO_sw, After PTO, BUW Closed //Control bit
	        "Console_In".Slot1.Ch1 := 1; //TDAuxSw
	        "Console_In".Slot1.Ch3 := 0; //TDEnableSw 
	END_IF;
	
	//TD Enable, ready to run
	IF #Test_Mode = #TDEnableMode OR #Test_Mode =#BUWAutoClHoldingMode OR #Test_Mode=#BUWAutoClHoldingModeDone OR #Test_Mode= #MudSaverCloseMode OR #Test_Mode=#MudSaverOpenMode OR #Test_Mode=#MudSaverAutoMode OR
	    #Test_Mode=#QuillLockMode OR #Test_Mode=#QuillLockModeDone OR #Test_Mode = #"MudSaverPumpRuningMode-0" OR #Test_Mode=#"MudSaverPumpRuningMode-1"
	    OR #Test_Mode= #ElevOpenMode OR #Test_Mode=#ElevCloseMode THEN
	        "Console_In".Slot1.Ch1 := 0; //TDAuxSw
	        "Console_In".Slot1.Ch3 := 1; //TDEnableSw
	        "IO_Settings".ElevClSw := 0; //No Elevator
	        "HPU_In".Slot4.Ch9 := 0; //"ElevClFeedback" := 0;  //No
	        "Console_In".Slot2.Ch2 := 1; // "ElevClSw" := "Console_In".Slot2.Ch2;
	        "Console_In".Slot2.Ch0 := 0;//"ElevOpSw" := "Console_In".Slot2.Ch0;/
	    END_IF;
	
	    IF #Test_Mode = #BUWAutoClHoldingMode  THEN
	        //BUW AutoClose Hold 
	        //To Open BUW 
	        //#Counter := 1;
	        "Console_In".Slot1.Ch12 := 1; //"TDModeMUSpinSw" := "Console_In".Slot1.Ch12; this is key to hold
	        "Console_In".Slot1.Ch13 := 0; //"TDModeMUTorqSw" := "Console_In".Slot1.Ch12;
	        "Console_In".Slot1.Ch14 := 0; //"TDBOSw" := "Console_In".Slot1.Ch12;
	        "Console_In".Slot1.Ch9 := 0; // BUWClSw, close
	    //ELSIF #Counter =1 THEN
	       // "Console_In".Slot1.Ch9 := 0; //"BUWClSw",open 
	        //"Console_In".Slot1.Ch12 := 1; //"TDModeMUSpinSw" := "Console_In".Slot1.Ch12;
	    END_IF;
	    IF #Test_Mode = #BUWAutoClHoldingModeDone THEN
	        "Console_In".Slot1.Ch12 := 0; //"TDModeMUSpinSw" := "Console_In".Slot1.Ch12;
	        "Console_In".Slot1.Ch13 := 0; //"TDModeMUTorqSw" := "Console_In".Slot1.Ch12;
	        "Console_In".Slot1.Ch14 := 0; //"TDBOSw" := "Console_In".Slot1.Ch12;
	        "Console_In".Slot1.Ch9 := 0; // BUWClSw
	    END_IF;
	    
	    IF #Test_Mode = #QuillLockMode THEN //Have to first do a fake MUTorq
	        //QuillLock
	//1. make sure MUCycleDone. 2. move BUWClSw on, 3. PTO on 4.  BUWClSw to QuillLockSw 
	   
	        "HPU_In".Slot6.Ch0 := 12345;//TD Pressure Fwd
	        "HPU_In".Slot6.Ch1 := 12;//TD Pressure Rev
	//1.  Init and BUWClSw on
	         "Console_In".Slot2.Ch4 := 0;//PTO_sw
	         "Console_In".Slot1.Ch13 := 0;//"TDModeMUTorqSw":= "Console_In".Slot1.Ch13; //Chang
	         "Console_In".Slot1.Ch9 := 1; // BUWClSw       //change
	         "Console_In".Slot1.Ch8 := 0; //Quill lock     //change
	//2.         
	        // "Console_In".Slot2.Ch4 := 1;//PTO_sw,  switch PTO to trigger
	           
	//3         
	        // "Console_In".Slot1.Ch9 := 0; // BUWClSw       //change
	        //  "Console_In".Slot1.Ch8 := 1; //Quill lock     //change
	         
	
	        END_IF;
	        IF #Test_Mode = #QuillLockModeDone THEN
	            
	            "Console_In".Slot1.Ch13 := 0;//"TDModeMUTorqSw":= "Console_In".Slot1.Ch13;
	            "Console_In".Slot1.Ch14 := 0; //"TDModeDrillRevSw
	            "Console_In".Slot1.Ch15 := 0; //"TDBOBeakOutSw" := "Console_In".Slot1.Ch15;
	            "HPU_In".Slot6.Ch0 := 12345;//TD Pressure Fwd
	            "HPU_In".Slot6.Ch1 := 12;//TD Pressure Rev
	
	            "Console_In".Slot2.Ch4 := 0;//PTO_sw
	            "Console_In".Slot1.Ch9 := 0; // BUWClSw
	            "Console_In".Slot1.Ch8 := 0; //Quill lock
	        END_IF;
	    IF #Test_Mode = #ElevCloseMode THEN
	        //Elevator Close
	        "Console_In".Slot2.Ch4 := 0;//PTO_sw
	        "IO_Settings".ElevClSw := 0;
	        
	        "HPU_In".Slot4.Ch9 := 0; //"ElevClFeedback":="HPU_In".Slot4.Ch9;
	        "Console_In".Slot2.Ch2 := 1; // "ElevClSw" := "Console_In".Slot2.Ch2;
	        "Console_In".Slot2.Ch0 := 0;//"ElevOpSw" := "Console_In".Slot2.Ch0;
	    END_IF;
	    IF #Test_Mode = #ElevOpenMode THEN
	        //Elevator Open
	        "Console_In".Slot2.Ch4 := 1;//PTO_sw
	        "Console_In".Slot2.Ch2 := 0; // "ElevClSw" := "Console_In".Slot2.Ch2;
	        "Console_In".Slot2.Ch0 := 1;//"ElevOpSw" := "Console_In".Slot2.Ch0;
	    END_IF;
	
	     IF #Test_Mode = #MudSaverCloseMode THEN
	         //Mud Saver Valve
	         //Close,Aux, Open
	         "Console_In".Slot1.Ch7 := 0; // //MPRunning
	         "Console_In".Slot2.Ch6 := 1; //"MSVClSw" := "Console_In".Slot2.Ch6;
	         "Console_In".Slot2.Ch7 := 0; //"MSVAutoSw" := "Console_In".Slot2.Ch7;
	         "Console_In".Slot2.Ch8 := 0; //"MSVOpSw" := "Console_In".Slot2.Ch8;
	     END_IF;
	     IF #Test_Mode = #MudSaverOpenMode THEN
	         "Console_In".Slot1.Ch7 := 0; // //MPRunning
	         "Console_In".Slot2.Ch6 := 0; //"MSVClSw" := "Console_In".Slot2.Ch6;
	         "Console_In".Slot2.Ch7 := 0; //"MSVAutoSw" := "Console_In".Slot2.Ch7;
	         "Console_In".Slot2.Ch8 := 1; //"MSVOpSw" := "Console_In".Slot2.Ch8;
	     END_IF;
	     IF #Test_Mode=#MudSaverAutoMode THEN
	         "Console_In".Slot1.Ch7 := 0; // //MPRunning
	         "Console_In".Slot2.Ch6 := 0; //"MSVClSw" := "Console_In".Slot2.Ch6;
	         "Console_In".Slot2.Ch7 := 1; //"MSVAutoSw" := "Console_In".Slot2.Ch7;
	         "Console_In".Slot2.Ch8 := 0; //"MSVOpSw" := "Console_In".Slot2.Ch8;
	     END_IF;
	     IF #Test_Mode = #"MudSaverPumpRuningMode-0" THEN
	         "Console_In".Slot1.Ch7 := 0; // //MPRunning
	         "Console_In".Slot2.Ch6 := 0; //"MSVClSw" := "Console_In".Slot2.Ch6;
	         "Console_In".Slot2.Ch7 := 1; //"MSVAutoSw" := "Console_In".Slot2.Ch7;
	         "Console_In".Slot2.Ch8 := 0; //"MSVOpSw" := "Console_In".Slot2.Ch8;
	     END_IF;
	     IF #Test_Mode = #"MudSaverPumpRuningMode-1" THEN
	         "Console_In".Slot1.Ch7 := 1; // //MPRunning
	         "Console_In".Slot2.Ch6 := 0; //"MSVClSw" := "Console_In".Slot2.Ch6;
	         "Console_In".Slot2.Ch7 := 1; //"MSVAutoSw" := "Console_In".Slot2.Ch7;
	         "Console_In".Slot2.Ch8 := 0; //"MSVOpSw" := "Console_In".Slot2.Ch8;
	     END_IF;
	//LEDs
	#PTOLED := "PTOLED"; //"Console_Out".Slot4.Ch0 := "PTOLED";
	#HpuFaultLed := "HPUFaultLED";//"Console_Out".Slot4.Ch1 := "HPUFaultLED";
	#BUWCLLED := "BUWClLED";
	#QuillLockLED := "QuillLockLED";
	#TDEnableLed := "TDEnLED";
	#MSVClLED := "MSVClLED";
	#ElevatorCLLED := "ElevClLED";
	//"Console_Out".Slot4.Ch2 := "TDFlushFaultLED";
	//"Console_Out".Slot4.Ch3 := "BUWClLED";
	//"Console_Out".Slot4.Ch4 := "TDEnLED";
	//"Console_Out".Slot4.Ch5 := "ConLowPurgeLED";
	//"Console_Out".Slot4.Ch6 := "MSVClLED";
	//"Console_Out".Slot4.Ch7 := "QuillLockLED";
	//"Console_Out".Slot4.Ch8 := "ElevClLED";
	//"Console_Out".Slot4.Ch9 := "Horn";
	//"Console_Out".Slot4.Ch10 := "MSVClInt";
	//"Console_Out".Slot4.Ch11 := "BUWClInt";
	//
	//Setup of TD Drive for all feedback signals
	//
	"Console_In".Slot3.Ch0 := 1000;//"MUTorqPotRaw":="Console_In".Slot3.Ch0;
	"Console_In".Slot3.Ch1 := 1100; //"DrillTorqPotRaw" := "Console_In".Slot3.Ch1;
	"Console_In".Slot3.Ch2 := 1200;;//"DrillThrottlePotRaw":="Console_In".Slot3.Ch2;
	
	//"Console_In".Slot1.Ch13 := 0;//"TDModeMUTorqSw":= "Console_In".Slot1.Ch13;
	//"Console_In".Slot1.Ch14 := 0; //"TDModeDrillRevSw
	//"Console_In".Slot1.Ch15 := 0; //"TDBOBeakOutSw" := "Console_In".Slot1.Ch15;
	
	"HPU_In".Slot2.COUNT_VALUE:=1000; //"RotaryCounts" := "HPU_In".Slot2.COUNT_VALUE;
	
	"HPU_In".Slot4.Ch0 := 1;   //"TankLowLevelSw" := "HPU_In".Slot4.Ch0;
	"HPU_In".Slot4.Ch1 := 1;   //"TankHighTempSw" := "HPU_In".Slot4.Ch1;
	
	"HPU_In".Slot4.Ch2 := 1;   //"TDFwdFilter1" := "HPU_In".Slot4.Ch2;
	"HPU_In".Slot4.Ch3 := 1;//"TDFwdFilter2" := "HPU_In".Slot4.Ch3;
	"HPU_In".Slot4.Ch4 := 1;//"TDRevFilter1" := "HPU_In".Slot4.Ch4;
	"HPU_In".Slot4.Ch5 := 1;//"TDRevFilter2" := "HPU_In".Slot4.Ch5;
	"HPU_In".Slot4.Ch6 := 1;//"AuxReturnFilter" := "HPU_In".Slot4.Ch6;
	
	"HPU_In".Slot5.Ch0 := 10000;//M1 Current
	"HPU_In".Slot5.Ch1 := 15000;//M2 Current
	IF #Test_Mode <> #QuillLockMode THEN
	    "HPU_In".Slot6.Ch0 := 12345;//TD Pressure Fwd
	    "HPU_In".Slot6.Ch1 := 12345;//TD Pressure Rev
	END_IF;
	"HPU_In".Slot6.Ch2 := 15000;  //"ClosedLoopTempRaw" := "HPU_In".Slot6.Ch2;
	"HPU_In".Slot6.Ch3 := 15000;  //Charge Flow
	"HPU_In".Slot6.Ch4 := 15000;  //Hot Oil Shuttle Flow
	"HPU_In".Slot6.Ch5 := 15000;  //Auxilliary Flow
	"HPU_In".Slot6.Ch6 := 15000;  //Charge Pressure1
	"HPU_In".Slot6.Ch7 := 15000;  //Charge Pressure2
	
	"HPU_In".Slot3.Ch0 := 1; //AuxPumpRunning feedback
	"HPU_In".Slot3.Ch1 := 1; //"CoolingFanRunning" := "HPU_In".Slot3.Ch1;
	
	
	IF #Test_Mode = #AuxByPassMode OR #Test_Mode = #AuxByPassModeDone THEN
	    "HPU_In".Slot3.Ch2 := 0;//M1Running
	    "HPU_In".Slot3.Ch3 := 0;//M2Running
	ELSE
	    "HPU_In".Slot3.Ch2 := 1;//M1Running
	    "HPU_In".Slot3.Ch3 := 1;//M2Running
	END_IF;
	"HPU_In".Slot3.Ch6 := 1;//M1HOA
	"HPU_In".Slot3.Ch7 := 1; //M2HOA
	"HPU_In".Slot3.Ch8 := 1;//"TDFlushFlowSw":="HPU_In".Slot3.Ch8; //blink the TEEnable LED
	"HPU_In".Slot3.Ch5 := 1; //"CoolingFanHOA" := "HPU_In".Slot3.Ch5;
	"HPU_In".Slot3.Ch4 := 1;//"AuxPumpHOA" := "HPU_In".Slot3.Ch4;
END_FUNCTION_BLOCK

ORGANIZATION_BLOCK "RPM"
{ S7_Optimized_Access := 'TRUE' }
VERSION : 0.1
   VAR_TEMP 
      CalcSpeedRPM : Real;
      Count_Per_Sec : Real;
   END_VAR


BEGIN
	#CalcSpeedRPM := ABS(DINT_TO_REAL("RotaryCounts" - "LastCount"));
	"LastCount" := "RotaryCounts";
	#Count_Per_Sec := INT_TO_REAL("Settings".RotEncPPR);
	IF "RotaryRPM" > 100 THEN
	    #CalcSpeedRPM := 1.0 * #CalcSpeedRPM / #Count_Per_Sec * 60.0 / 1.0;
	ELSIF "RotaryRPM" > 55.0 THEN
	    #CalcSpeedRPM := 1.0 * #CalcSpeedRPM / #Count_Per_Sec * 60.0 / 1.0;
	ELSE
	    #CalcSpeedRPM := 1.0 * #CalcSpeedRPM / #Count_Per_Sec * 60.0 / 1.0;
	END_IF;
	"RotaryRPMActual" := ABS(#CalcSpeedRPM);
	"LowPassFilter_DB"(InputSignal := ABS(#CalcSpeedRPM),
	                   Alpha := 0.7,
	                   FilteredSignal => "RotaryRPM");
END_ORGANIZATION_BLOCK

FUNCTION "Unused IO Ports" : Void
{ S7_Optimized_Access := 'TRUE' }
VERSION : 0.1

BEGIN
	
	//Rig 3 unused IO Port. Set its value to ).
	"ClosedLoopTempCFilt" := 0;
	"ClosedLoopTempCMax" := 0;
	"HotOilFlowGPMFilt" := 0;
	"AuxFlowGPMFilt" := 0;
	"ChargeFlowGPMFilt" := 0;
	"ChargePress1PSIFilt" := 0;
	"ChargePress2PSIFilt" := 0;
END_FUNCTION

FUNCTION "TM_Pulse_mA2Raw" : Int
{ S7_Optimized_Access := 'TRUE' }
VERSION : 0.1
   VAR_INPUT 
      maInput : Real;
   END_VAR


BEGIN
	(* TM_Pulse_mA2Raw Written BY Kristopher Gimenez January 19,2023
	This block is used to convert the ma current outputs to a raw signal for  2CH TM pulse module. Note 2A = 27648. 
	*)
	
	
	#TM_Pulse_mA2Raw := REAL_TO_INT(#maInput/2000*27648);
	
END_FUNCTION

FUNCTION "MapRemConsoleOutputs" : Void
{ S7_Optimized_Access := 'TRUE' }
VERSION : 0.1

BEGIN
	(* #MapConsoleOutputs Written BY Kristopher Gimenez January 23,2023
	This block is will map the output variables and convert raw signals into measured values
	*)
	
	
	
	//Slot 4 16x Digital Outputs
	"RemConsole_Out".PTOLED:="PTOLED";
	"RemConsole_Out".HPUFaultLED := "HPUFaultLED";
	"RemConsole_Out".TDFaultLED := "TDFlushFaultLED";
	"RemConsole_Out".BUWClLED := "BUWClLED";
	"RemConsole_Out".TDEnLED := "TDEnLED";
	"RemConsole_Out".MSVClLED := "MSVClLED";
	"RemConsole_Out".QuillLockedLED:= "QuillLockLED";
	"RemConsole_Out".ElevClLED:= "ElevClLED";
	"RemConsole_Out".Horn := "Horn";
	"RemConsole_Out".MSVClInt:= "MSVClInt";
	"RemConsole_Out".BUWClInt := "BUWClInt";
	(*Spare Outputs
	"Console_Out".Slot4.Ch12 := ;
	"Console_Out".Slot4.Ch13 := ;
	"Console_Out".Slot4.Ch14 := ;
	"Console_Out".Slot4.Ch15 := ;
	*)
	
	
	
	
	//Slot 5 4 x AQ U/I
	"AoUI_Scaling"(Measured:="DrillRecTorqFtLbs",
	               Max:=40000.0,
	               Min:=0,
	               s7Raw=>"DrillRecTorqRaw",
	               mAOutput=>"DrillRecTorqmA"); //4-20ma = 0-40 000 ft-lbs
	"AoUI_Scaling"(Measured:="DrillRecRPM",
	               Max:=200.0,
	               Min:=0,
	               s7Raw=>"DrillRecRPMRaw",
	               mAOutput=>"DrillRecRPMmA");// 4-20ma = 0-200 RPM
	
	
	"RemConsole_Out".DrillRecTorq := "DrillRecTorqRaw";
	"RemConsole_Out".DrillRecRPM := "DrillRecRPMRaw";
END_FUNCTION

DATA_BLOCK "Alarms_DB"   // DB9
// stored: InstanceOfName Alarms, InstanceOfType FB
"Alarms"
BEGIN
END_DATA_BLOCK

DATA_BLOCK "Block_1_DB_2"   // DB36
// stored: InstanceOfName Block_1, InstanceOfType FB
"Block_1"
BEGIN
END_DATA_BLOCK

DATA_BLOCK "Comms_DB"   // DB22
// stored: AutoNumber false, InstanceOfName Comms, InstanceOfType FB
"Comms"
BEGIN
END_DATA_BLOCK

DATA_BLOCK "LowPassFilter_DB"   // DB4
// stored: InstanceOfName LowPassFilter, InstanceOfType FB
"LowPassFilter"
BEGIN
END_DATA_BLOCK

DATA_BLOCK "Aux_Functions_DB"   // DB16
// stored: AutoNumber false, InstanceOfName Aux_Functions, InstanceOfType FB
"Aux_Functions"
BEGIN
END_DATA_BLOCK

DATA_BLOCK "Aux_Motor_Control_DB"   // DB12
// stored: AutoNumber false, InstanceOfName Aux_Motor_Control, InstanceOfType FB
"Aux_Motor_Control"
BEGIN
END_DATA_BLOCK

DATA_BLOCK "Calculations_DB"   // DB10
// stored: AutoNumber false, InstanceOfName Calculations, InstanceOfType FB
"Calculations"
BEGIN
END_DATA_BLOCK

DATA_BLOCK "HMI_DB"   // DB20
// stored: AutoNumber false, InstanceOfName HMI, InstanceOfType FB
"HMI"
BEGIN
   DHScreen[0..4] := 0;
   HPUScreen[0..1] := 1;
   HPUScreen[2] := 0;
   HPUScreen[3] := 1;
   HPUScreen[4] := 0;
   ConsoleScreen[0..1] := 1;
   ConsoleScreen[2] := 0;
   ConsoleScreen[3] := 1;
   ConsoleScreen[4] := 0;
   LampTestLamp_TP.PT := T#0MS;
   LampTestLamp_TP.IN := FALSE;
   LampTestHorn_TP.PT := T#0MS;
   LampTestHorn_TP.IN := FALSE;
   HornSilence_TOF.PT := T#0MS;
   HornSilence_TOF.IN := FALSE;
   Alarms1_To_Unified[0..15] := FALSE;
   Alarms2_To_Unified[0..5] := FALSE;
   Alarms2_To_Unified[6..9] := TRUE;
   Alarms2_To_Unified[10] := FALSE;
   Alarms2_To_Unified[11..12] := TRUE;
   Alarms2_To_Unified[13..15] := FALSE;
   Warnings1_To_Unified[0] := TRUE;
   Warnings1_To_Unified[1..15] := FALSE;
END_DATA_BLOCK

DATA_BLOCK "LEDS_DB"   // DB17
// stored: AutoNumber false, InstanceOfName LEDS, InstanceOfType FB
"LEDS"
BEGIN
END_DATA_BLOCK

DATA_BLOCK "RotPosCalc_DB"   // DB11
// stored: AutoNumber false, InstanceOfName Rot_Pos_Calc, InstanceOfType FB
"Rot_Pos_Calc"
BEGIN
END_DATA_BLOCK

DATA_BLOCK "System_Enable_DB"   // DB15
// stored: AutoNumber false, InstanceOfName System_Enable, InstanceOfType FB
"System_Enable"
BEGIN
END_DATA_BLOCK

DATA_BLOCK "TD_Control_DB"   // DB19
// stored: AutoNumber false, InstanceOfName TD_Control, InstanceOfType FB
"TD_Control"
BEGIN
END_DATA_BLOCK

DATA_BLOCK "TD_Start_CAT_DB"   // DB14
// stored: AutoNumber false, InstanceOfName TD_Motor_Start_CAT, InstanceOfType FB
"TD_Motor_Start_CAT"
BEGIN
END_DATA_BLOCK

DATA_BLOCK "TD_Start_Elec_DB"   // DB13
// stored: AutoNumber false, InstanceOfName TD_Motor_Start_Elec, InstanceOfType FB
"TD_Motor_Start_Elec"
BEGIN
END_DATA_BLOCK

DATA_BLOCK "Timers_DB"   // DB21
// stored: AutoNumber false, InstanceOfName Timers, InstanceOfType FB
"Timers"
BEGIN
END_DATA_BLOCK

DATA_BLOCK "BO_Torq_DB"   // DB33
// stored: AutoNumber false, InstanceOfName BO_Torq, InstanceOfType FB
"BO_Torq"
BEGIN
END_DATA_BLOCK

DATA_BLOCK "Drill_DB"   // DB30
// stored: AutoNumber false, InstanceOfName Drill, InstanceOfType FB
"Drill"
BEGIN
END_DATA_BLOCK

DATA_BLOCK "MU_Spin_DB"   // DB31
// stored: AutoNumber false, InstanceOfName MU_Spin, InstanceOfType FB
"MU_Spin"
BEGIN
END_DATA_BLOCK

DATA_BLOCK "MU_Torq_DB"   // DB32
// stored: AutoNumber false, InstanceOfName MU_Torq, InstanceOfType FB
"MU_Torq"
BEGIN
END_DATA_BLOCK

DATA_BLOCK "Oscilate_DB"   // DB34
// stored: AutoNumber false, InstanceOfName Oscillate, InstanceOfType FB
"Oscillate"
BEGIN
END_DATA_BLOCK

DATA_BLOCK "CoolingFanOffTON"   // DB29
{ S7_Optimized_Access := 'TRUE' }
// stored: InstanceOfName IEC_TIMER, OfSystemLibElement IEC_TIMER, OfSystemLibVersion 1.0
"IEC_TIMER"
   // VAR
   //    PT : Time;
   //    ET { ExternalWritable := 'False'} : Time;
   //    IN : Bool;
   //    Q { ExternalWritable := 'False'} : Bool;
   // END_VAR
BEGIN
END_DATA_BLOCK

DATA_BLOCK "ElevCl_TON_10s"   // DB3
{ S7_Optimized_Access := 'TRUE' }
// stored: InstanceOfName IEC_TIMER, OfSystemLibElement IEC_TIMER, OfSystemLibVersion 1.0
"IEC_TIMER"
   // VAR
   //    PT : Time;
   //    ET { ExternalWritable := 'False'} : Time;
   //    IN : Bool;
   //    Q { ExternalWritable := 'False'} : Bool;
   // END_VAR
BEGIN
END_DATA_BLOCK

DATA_BLOCK "IEC_Timer_0_DB"   // DB2
{ S7_Optimized_Access := 'TRUE' }
// stored: InstanceOfName IEC_TIMER, OfSystemLibElement IEC_TIMER, OfSystemLibVersion 1.0
"IEC_TIMER"
   // VAR
   //    PT : Time;
   //    ET { ExternalWritable := 'False'} : Time;
   //    IN : Bool;
   //    Q { ExternalWritable := 'False'} : Bool;
   // END_VAR
BEGIN
END_DATA_BLOCK

DATA_BLOCK "IEC_Timer_0_DB_1"   // DB5
{ S7_Optimized_Access := 'TRUE' }
// stored: InstanceOfName IEC_TIMER, OfSystemLibElement IEC_TIMER, OfSystemLibVersion 1.0
"IEC_TIMER"
   // VAR
   //    PT : Time;
   //    ET { ExternalWritable := 'False'} : Time;
   //    IN : Bool;
   //    Q { ExternalWritable := 'False'} : Bool;
   // END_VAR
BEGIN
END_DATA_BLOCK

DATA_BLOCK "IEC_Timer_0_DB_10"   // DB27
{ S7_Optimized_Access := 'TRUE' }
// stored: InstanceOfName IEC_TIMER, OfSystemLibElement IEC_TIMER, OfSystemLibVersion 1.0
"IEC_TIMER"
   // VAR
   //    PT : Time;
   //    ET { ExternalWritable := 'False'} : Time;
   //    IN : Bool;
   //    Q { ExternalWritable := 'False'} : Bool;
   // END_VAR
BEGIN
END_DATA_BLOCK

DATA_BLOCK "IEC_Timer_0_DB_11"   // DB28
{ S7_Optimized_Access := 'TRUE' }
// stored: InstanceOfName IEC_TIMER, OfSystemLibElement IEC_TIMER, OfSystemLibVersion 1.0
"IEC_TIMER"
   // VAR
   //    PT : Time;
   //    ET { ExternalWritable := 'False'} : Time;
   //    IN : Bool;
   //    Q { ExternalWritable := 'False'} : Bool;
   // END_VAR
BEGIN
END_DATA_BLOCK

DATA_BLOCK "IEC_Timer_0_DB_2"   // DB6
{ S7_Optimized_Access := 'TRUE' }
// stored: InstanceOfName IEC_TIMER, OfSystemLibElement IEC_TIMER, OfSystemLibVersion 1.0
"IEC_TIMER"
   // VAR
   //    PT : Time;
   //    ET { ExternalWritable := 'False'} : Time;
   //    IN : Bool;
   //    Q { ExternalWritable := 'False'} : Bool;
   // END_VAR
BEGIN
END_DATA_BLOCK

DATA_BLOCK "IEC_Timer_0_DB_3"   // DB7
{ S7_Optimized_Access := 'TRUE' }
// stored: InstanceOfName IEC_TIMER, OfSystemLibElement IEC_TIMER, OfSystemLibVersion 1.0
"IEC_TIMER"
   // VAR
   //    PT : Time;
   //    ET { ExternalWritable := 'False'} : Time;
   //    IN : Bool;
   //    Q { ExternalWritable := 'False'} : Bool;
   // END_VAR
BEGIN
END_DATA_BLOCK

DATA_BLOCK "IEC_Timer_0_DB_4"   // DB8
{ S7_Optimized_Access := 'TRUE' }
// stored: InstanceOfName IEC_TIMER, OfSystemLibElement IEC_TIMER, OfSystemLibVersion 1.0
"IEC_TIMER"
   // VAR
   //    PT : Time;
   //    ET { ExternalWritable := 'False'} : Time;
   //    IN : Bool;
   //    Q { ExternalWritable := 'False'} : Bool;
   // END_VAR
BEGIN
END_DATA_BLOCK

DATA_BLOCK "IEC_Timer_0_DB_5"   // DB18
{ S7_Optimized_Access := 'TRUE' }
// stored: InstanceOfName IEC_TIMER, OfSystemLibElement IEC_TIMER, OfSystemLibVersion 1.0
"IEC_TIMER"
   // VAR
   //    PT : Time;
   //    ET { ExternalWritable := 'False'} : Time;
   //    IN : Bool;
   //    Q { ExternalWritable := 'False'} : Bool;
   // END_VAR
BEGIN
END_DATA_BLOCK

DATA_BLOCK "IEC_Timer_0_DB_6"   // DB23
{ S7_Optimized_Access := 'TRUE' }
// stored: InstanceOfName IEC_TIMER, OfSystemLibElement IEC_TIMER, OfSystemLibVersion 1.0
"IEC_TIMER"
   // VAR
   //    PT : Time;
   //    ET { ExternalWritable := 'False'} : Time;
   //    IN : Bool;
   //    Q { ExternalWritable := 'False'} : Bool;
   // END_VAR
BEGIN
END_DATA_BLOCK

DATA_BLOCK "IEC_Timer_0_DB_7"   // DB24
{ S7_Optimized_Access := 'TRUE' }
// stored: InstanceOfName IEC_TIMER, OfSystemLibElement IEC_TIMER, OfSystemLibVersion 1.0
"IEC_TIMER"
   // VAR
   //    PT : Time;
   //    ET { ExternalWritable := 'False'} : Time;
   //    IN : Bool;
   //    Q { ExternalWritable := 'False'} : Bool;
   // END_VAR
BEGIN
END_DATA_BLOCK

DATA_BLOCK "IEC_Timer_0_DB_8"   // DB25
{ S7_Optimized_Access := 'TRUE' }
// stored: InstanceOfName IEC_TIMER, OfSystemLibElement IEC_TIMER, OfSystemLibVersion 1.0
"IEC_TIMER"
   // VAR
   //    PT : Time;
   //    ET { ExternalWritable := 'False'} : Time;
   //    IN : Bool;
   //    Q { ExternalWritable := 'False'} : Bool;
   // END_VAR
BEGIN
END_DATA_BLOCK

DATA_BLOCK "IEC_Timer_0_DB_9"   // DB26
{ S7_Optimized_Access := 'TRUE' }
// stored: InstanceOfName IEC_TIMER, OfSystemLibElement IEC_TIMER, OfSystemLibVersion 1.0
"IEC_TIMER"
   // VAR
   //    PT : Time;
   //    ET { ExternalWritable := 'False'} : Time;
   //    IN : Bool;
   //    Q { ExternalWritable := 'False'} : Bool;
   // END_VAR
BEGIN
END_DATA_BLOCK
